TYPE Robot :
STRUCT
	JointStates 	: JointState;		// STRUCT to contain all of the joint states (pos,vel,I)
	Job         	: UINT := 0;		// Job the robot should be performing
	Active      	: BOOL := FALSE;	// Status bit - TRUE if robot is moving
	Transfer		: BOOL := FALSE;	// Status bit - (Robot1 is ready to transfer)
END_STRUCT
END_TYPE

(* stored: Version 1.1.0.1, ProductVersion 3.1.0.36
   DUT Robot: Id {dd225ca7-9894-4635-b155-bb1b723c9fa8} *)
